Universal Robots PolyScope program: cottonFill.urp

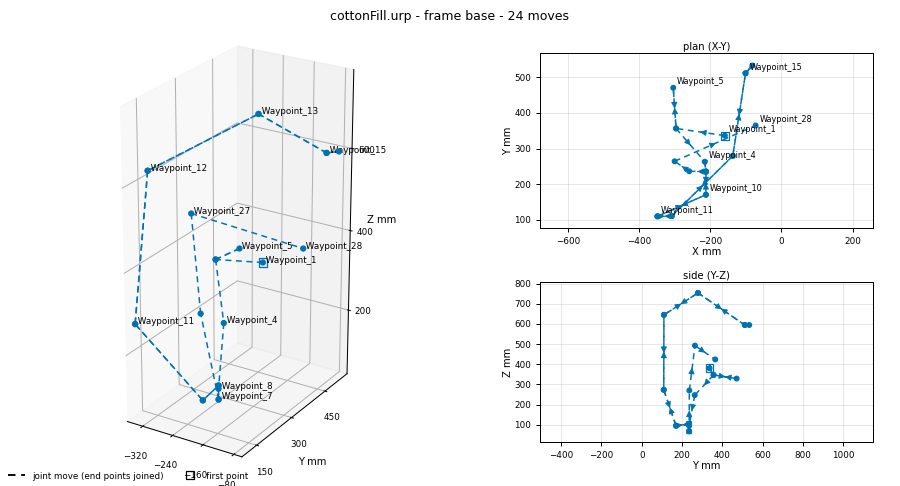
[picture p0: tool path of cottonFill.urp in frame base, 24 of 26 moves have a stored position in this frame; points joined in program order, loops and branches not executed]
Program cottonFill (installation=default directory=/programs/DavidMelin createdIn=5.12.4.1101661 lastSavedIn=5.12.4.1101661 robotSerialNumber=20225502378)
Calibrated DH parameters: a=[0.00022, -0.425328, -0.389701, 0.000059, 0.000065, 0]; d=[0.162608, 0.803456, 9.992211, -10.662202, 0.099702, 0.099559]; alpha=[1.570756, 0.001543, 0.004316, 1.570651, -1.570122, 0]; deltaTheta=[0, 0.002917, 0.116094, -0.119008, 0, -0.000001]
Robot Program (runOnlyOnce=true)
  MoveJ speed 60 deg/s, acceleration 80 deg/s^2 (useActiveTCP=true) feature=Base
    Waypoint Waypoint (Variable): variable=cotonHomePos
  URCap Gripper (Robotiq_Grippers, Robotiq Inc.) dataModel(position=0.0, force=0.0, speed=0.0, positionInDouble=0.0, forceInDouble=0.0, speedInDouble=0.0, slaveIds=[9], blocking=true)
  MoveJ speed 60 deg/s, acceleration 80 deg/s^2 (useActiveTCP=true) feature=Base
    Waypoint Waypoint_1: TCP in base x=-158.969 y=336.336 z=379.953 mm, rx=-2.2924 ry=-1.1159 rz=-0.9813 rad; joints [149.291, -67.032, -128.013, -78.577, 42.37, 8.935] deg
    Waypoint Waypoint_2: TCP in base x=-296.185 y=356.475 z=346.661 mm, rx=-1.2462 ry=-1.1782 rz=-1.1663 rad; joints [159.144, -90.902, -110.13, -161.705, -20.728, 95.682] deg
    Waypoint Waypoint_5: TCP in base x=-304.046 y=470.843 z=328.792 mm, rx=-1.2851 ry=-1.1466 rz=-1.1584 rad; joints [145.798, -103.932, -97.829, -160.878, -32.585, 97.219] deg
  URCap Gripper (Robotiq_Grippers, Robotiq Inc.) dataModel(position=40.0, force=100.0, speed=50.0, positionInDouble=40.0, forceInDouble=100.0, speedInDouble=50.0, slaveIds=[9], blocking=true)
  Wait Sleep waitTime=0.5
  URCap Gripper (Robotiq_Grippers, Robotiq Inc.) dataModel(position=0.0, force=50.0, speed=0.0, positionInDouble=0.0, forceInDouble=50.0, speedInDouble=0.0, slaveIds=[9], blocking=true)
  MoveJ speed 60 deg/s, acceleration 80 deg/s^2 (useActiveTCP=true) feature=Base
    Waypoint Waypoint_3: TCP in base x=-296.186 y=356.48 z=346.657 mm, rx=-1.2461 ry=-1.1782 rz=-1.1663 rad; joints [159.144, -90.903, -110.13, -161.705, -20.729, 95.68] deg
    Waypoint Waypoint_4: TCP in base x=-215.345 y=262.93 z=246.585 mm, rx=-1.5529 ry=0.0723 rz=0.0204 rad; joints [172.692, -77.601, -139.149, -135.1, -5.393, 175.311] deg
    Waypoint Waypoint_8: TCP in base x=-212.222 y=235.158 z=94.662 mm, rx=-1.5611 ry=0.0422 rz=-0.0025 rad; joints [179.619, -108.568, -145.288, -123.216, 1.457, 198.52] deg
    Waypoint Waypoint_7: TCP in base x=-212.2 y=235.152 z=67.602 mm, rx=-1.5607 ry=0.0534 rz=-0.014 rad; joints [179.594, -113.921, -146.687, -110.828, 2.26, 192.873] deg
  URCap Gripper (Robotiq_Grippers, Robotiq Inc.) dataModel(position=100.0, force=100.0, speed=100.0, positionInDouble=100.0, forceInDouble=100.0, speedInDouble=100.0, slaveIds=[9], blocking=true)
  MoveJ speed 60 deg/s, acceleration 80 deg/s^2 (useActiveTCP=true) feature=Base
    Waypoint Waypoint_9: TCP in base x=-212.191 y=235.153 z=103.019 mm, rx=-1.5607 ry=0.0534 rz=-0.0141 rad; joints [179.602, -105.429, -146.39, -119.086, 2.247, 192.34] deg
    Waypoint Waypoint_10: TCP in base x=-212.225 y=170.121 z=94.663 mm, rx=-1.5611 ry=0.0422 rz=-0.0025 rad; joints [198.138, -103.436, -154.021, -103.885, 19.93, 182.683] deg
    Waypoint Waypoint_11: TCP in base x=-348.674 y=109.325 z=273.015 mm, rx=-1.7492 ry=0.4046 rz=-0.13 rad; joints [198.175, -87.425, -123.219, -128.259, 38.368, 170.849] deg
    Waypoint Waypoint_12: TCP in base x=-308.362 y=110.06 z=644.877 mm, rx=-1.8267 ry=0.394 rz=-0.3883 rad; joints [198.159, -82.226, -70.41, -185.501, 48.305, 161.054] deg
    Waypoint Waypoint_13: TCP in base x=-136.648 y=279.266 z=753.567 mm, rx=-2.0676 ry=0.2393 rz=-0.6153 rad; joints [161.273, -73.285, -62.138, -163.751, 30.284, 101.182] deg
    Waypoint Waypoint_15: TCP in base x=-100.834 y=511.599 z=594.425 mm, rx=-2.2262 ry=0.3336 rz=-0.5673 rad; joints [125.103, -85.839, -90.205, -71.687, 39.214, 41.384] deg
    Waypoint Waypoint_16: TCP in base x=-81.571 y=533.408 z=594.553 mm, rx=-1.9075 ry=-1.8699 rz=-1.3955 rad; joints [121.728, -88.249, -89.284, -65.33, 39.685, -70.14] deg
    Waypoint Waypoint_17: TCP in base x=-100.83 y=511.612 z=594.407 mm, rx=-2.2262 ry=0.3336 rz=-0.5673 rad; joints [125.102, -85.841, -90.205, -71.688, 39.216, 41.384] deg
    Waypoint Waypoint_18: TCP in base x=-136.657 y=279.278 z=753.553 mm, rx=-2.0676 ry=0.2393 rz=-0.6154 rad; joints [161.27, -73.287, -62.139, -163.751, 30.284, 101.181] deg
    Waypoint Waypoint_19: TCP in base x=-308.344 y=110.069 z=644.886 mm, rx=-1.8267 ry=0.3941 rz=-0.3883 rad; joints [198.158, -82.224, -70.41, -185.5, 48.306, 161.054] deg
    Waypoint Waypoint_20: TCP in base x=-348.671 y=109.339 z=273.013 mm, rx=-1.7492 ry=0.4046 rz=-0.13 rad; joints [198.173, -87.426, -123.219, -128.26, 38.366, 170.849] deg
    Waypoint Waypoint_24: TCP in base x=-212.231 y=170.125 z=94.66 mm, rx=-1.5611 ry=0.0423 rz=-0.0025 rad; joints [198.136, -103.438, -154.02, -103.884, 19.929, 182.682] deg
    Waypoint Waypoint_25: TCP in base x=-212.178 y=235.144 z=103.015 mm, rx=-1.5607 ry=0.0533 rz=-0.0141 rad; joints [179.604, -105.429, -146.392, -119.087, 2.248, 192.339] deg
    Waypoint Waypoint_6: TCP in base x=-212.215 y=235.14 z=67.605 mm, rx=-1.5607 ry=0.0534 rz=-0.014 rad; joints [179.597, -113.921, -146.686, -110.828, 2.26, 192.872] deg
  URCap Gripper (Robotiq_Grippers, Robotiq Inc.) dataModel(position=0.0, force=0.0, speed=0.0, positionInDouble=0.0, forceInDouble=0.0, speedInDouble=0.0, slaveIds=[9], blocking=true)
  MoveJ speed 60 deg/s, acceleration 80 deg/s^2 (useActiveTCP=true) feature=Base
    Waypoint Waypoint_26: TCP in base x=-259.242 y=236.183 z=269.664 mm, rx=-1.5587 ry=0.0885 rz=0.0371 rad; joints [179.506, -85.218, -129.18, -160.168, 1.474, 199.152] deg
    Waypoint Waypoint_27: TCP in base x=-300.189 y=264.127 z=492.253 mm, rx=-1.3159 ry=2.6876 rz=0.6162 rad; joints [163.651, -69.69, -110.363, -77.407, 69.871, 199.152] deg
    Waypoint Waypoint_28: TCP in base x=-72.415 y=364.804 z=423.589 mm, rx=0.5179 ry=-2.985 rz=-0.1444 rad; joints [121.305, -69.141, -118.356, -75.185, 94.013, 191.802] deg
    Waypoint Waypoint (Variable): variable=cotonHomePos
